FUNCTION_BLOCK CAT_Jacks (* Composite Function Block Type *)
  (* Standard: 61499-2 *)
  (* Version 0.0, 15/09/2021, Pranay Jhunjhunwala, Schneider Electric, template *)
  PACKAGE Main;
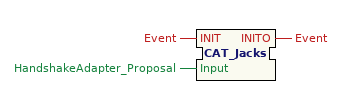
  EVENT_INPUT
    INIT; (* Initialization Request *)
  END_EVENT
  EVENT_OUTPUT
    INITO; (* Initialization Confirm *)
  END_EVENT
  SOCKETS
    Input : HandshakeAdapter_Proposal;
  END_SOCKETS
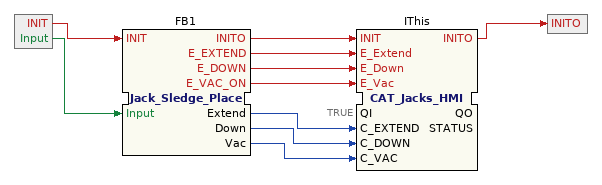
  FBS
    FB1 : Jack_Sledge_Place;
    IThis : CAT_Jacks_HMI(QI := TRUE);
  END_FBS
  EVENT_CONNECTIONS
    INIT TO FB1.INIT;
    FB1.INITO TO IThis.INIT;
    FB1.E_EXTEND TO IThis.E_Extend;
    FB1.E_DOWN TO IThis.E_Down;
    FB1.E_VAC_ON TO IThis.E_Vac;
    IThis.INITO TO INITO;
  END_CONNECTIONS
  DATA_CONNECTIONS
    FB1.Extend TO IThis.C_EXTEND;
    FB1.Down TO IThis.C_DOWN;
    FB1.Vac TO IThis.C_VAC;
  END_CONNECTIONS
  ADAPTER_CONNECTIONS
    Input TO FB1.Input;
  END_CONNECTIONS
END_FUNCTION_BLOCK
